{region '#Template'}
	{attribute 'Version' := '5.0.0.0'}
	{attribute 'Tags' := '"LCID": "1031", "Text": "Universal, Damper, Aggregate"'}
	{attribute 'Tags' := '"LCID": "1033", "Text": "Universal, Damper, Aggregate"'}
	{attribute 'Using' := '"Type": "Template", "URI": "EC_ID"'}
	{attribute 'Using' := '"Type": "Template", "URI": "BA2_Param"'}
	{attribute 'Description' := '"LCID": "1031", "Text": "2 Punkt Klappe mit Endlagenschalter"'}
	{attribute 'Description' := '"LCID": "1033", "Text": "2 point damper with limit switch"'}
{endregion}			 
FUNCTION_BLOCK FB_BA_Dmp2P EXTENDS FB_BA_ActuatorCmd
VAR_INPUT
END_VAR
VAR_OUTPUT
	bSwiOpn					: BOOL;
	bSwiCls					: BOOL;
END_VAR
VAR_INPUT CONSTANT
	SwiOpn					: FB_BA_BI_Raw;
	SwiCls					: FB_BA_BI_Raw;
	MonitOpen				: FB_BA_FdbBinary;
	MonitClose				: FB_BA_FdbBinary;
END_VAR	
VAR	
END_VAR

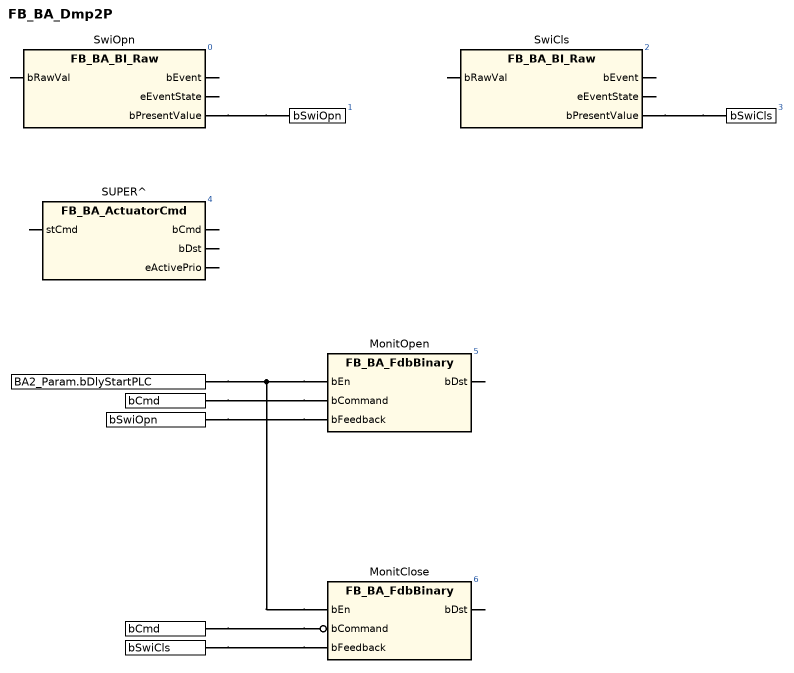
SwiOpn(); // FB_BA_BI_Raw
bSwiOpn := SwiOpn.bPresentValue;
SwiCls(); // FB_BA_BI_Raw
bSwiCls := SwiCls.bPresentValue;
SUPER^(); // FB_BA_ActuatorCmd
MonitOpen(bEn := BA2_Param.bDlyStartPLC, bCommand := bCmd, bFeedback := bSwiOpn); // FB_BA_FdbBinary
MonitClose(bEn := BA2_Param.bDlyStartPLC, bCommand := NOT bCmd, bFeedback := bSwiCls); // FB_BA_FdbBinary

METHOD FB_init : BOOL
VAR_INPUT
	bInitRetains : BOOL; // if TRUE, the retain variables are initialized (warm start / cold start)
	bInCopyCode : BOOL;  // if TRUE, the instance afterwards gets moved into the copy code (online change)
END_VAR
SwiOpn.iParent							:= THIS^;
SwiOpn.iLabel							:= LblFun_FeedbackOPEN;  
SwiOpn.sObjectName						:='{Idx=01}';
SwiOpn.ePolarity						:= E_BA_Polarity.eReverse;
SwiOpn.sActiveText 						:= txtEvent_Reached;
SwiOpn.sInactiveText 					:= txtEvent_NotReached;
SwiOpn.nEventClassID					:= EC_ID.NC80;
SwiOpn.stTimeDelay.nToNormal			:= BA2_Param.nDefTimeDelay_ToNormal;
SwiOpn.stTimeDelay.nToAbnormal			:= BA2_Param.nDefTimeDelay_ToAbnormal;
SwiOpn.bAlarmValue						:= TRUE;
SwiOpn.aEventTransitionText[1]			:= txtEvent_Active;
SwiOpn.aEventTransitionText[2]			:= txtEvent_None;
SwiOpn.aEventTransitionText[3]			:= txtEvent_Normal;
SwiOpn.bEventDetectionEnable			:= FALSE;
SwiOpn.eEnPlantLock						:= E_BA_LockPriority.eNoLock;	

SwiCls.iParent							:= THIS^;
SwiCls.iLabel							:= LblFun_FeedbackCLOSED; 
SwiCls.sObjectName						:='{Idx=01}';
SwiCls.ePolarity						:= E_BA_Polarity.eReverse;
SwiCls.sActiveText 						:= txtEvent_Reached;
SwiCls.sInactiveText 					:= txtEvent_NotReached;
SwiCls.nEventClassID					:= EC_ID.NC80;
SwiCls.stTimeDelay.nToNormal			:= BA2_Param.nDefTimeDelay_ToNormal;
SwiCls.stTimeDelay.nToAbnormal			:= BA2_Param.nDefTimeDelay_ToAbnormal;
SwiCls.bAlarmValue						:= TRUE;
SwiCls.aEventTransitionText[1]			:= txtEvent_Active;
SwiCls.aEventTransitionText[2]			:= txtEvent_None;
SwiCls.aEventTransitionText[3]			:= txtEvent_Normal;
SwiCls.bEventDetectionEnable			:= FALSE;
SwiCls.eEnPlantLock						:= E_BA_LockPriority.eNoLock;

MonitOpen.iParent						:= THIS^;
MonitOpen.iLabel						:= LblCtl_FeedbackMonitoring;  
MonitOpen.sObjectName					:='{Idx=01}';
MonitOpen.eDPADMode						:= E_BA_DPADMode.eIncludeDescription;
MonitOpen.DelayFeedback.fValueRm		:= 180.0;
MonitOpen.DelayFeedback.sObjectName		:='{Idx=01}';
MonitOpen.Dst.bEventDetectionEnable		:= TRUE;
MonitOpen.Dst.eEnPlantLock				:= E_BA_LockPriority.eLocalMedium;

MonitClose.iParent						:= THIS^;
MonitClose.iLabel						:= LblCtl_FeedbackMonitoring;
MonitClose.sObjectName					:='{Idx=02}';
MonitClose.eDPADMode					:= E_BA_DPADMode.eIncludeDescription;
MonitClose.DelayFeedback.fValueRm		:= 180.0;
MonitClose.DelayFeedback.iLabel			:= LblFun_FeedbackDelay;
MonitClose.DelayFeedback.sObjectName	:='{Idx=02}';
MonitClose.Dst.iLabel					:= LblFun_Fault;
MonitClose.Dst.sObjectName				:='{Idx=02}';
MonitClose.Dst.bEventDetectionEnable	:= TRUE;
MonitClose.Dst.eEnPlantLock				:= E_BA_LockPriority.eNoLock;
END_METHOD

END_FUNCTION_BLOCK

(* stored: Version 1.1.0.1, ProductVersion 3.1.4024.12
   POU FB_BA_Dmp2P: Id {dc19b11c-a8c9-4db0-aed4-7be89da624f7}, SpecialFunc None
   Method FB_init: Id {e6bcaade-5b65-465e-ab86-bc6abfdd6bfa} *)
